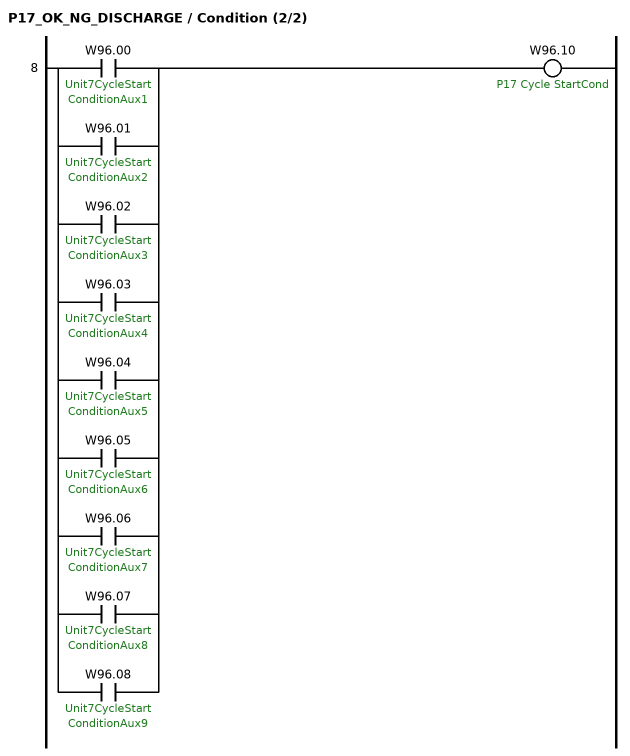
; [picture p288: P17_OK_NG_DISCHARGE / Condition, rungs 8-8]
; rung 8
LD W96.00  ; Unit7CycleStartConditionAux1
OR W96.01  ; Unit7CycleStartConditionAux2
OR W96.02  ; Unit7CycleStartConditionAux3
OR W96.03  ; Unit7CycleStartConditionAux4
OR W96.04  ; Unit7CycleStartConditionAux5
OR W96.05  ; Unit7CycleStartConditionAux6
OR W96.06  ; Unit7CycleStartConditionAux7
OR W96.07  ; Unit7CycleStartConditionAux8
OR W96.08  ; Unit7CycleStartConditionAux9
OUT W96.10  ; P17 Cycle StartCond

### Section Device_Output

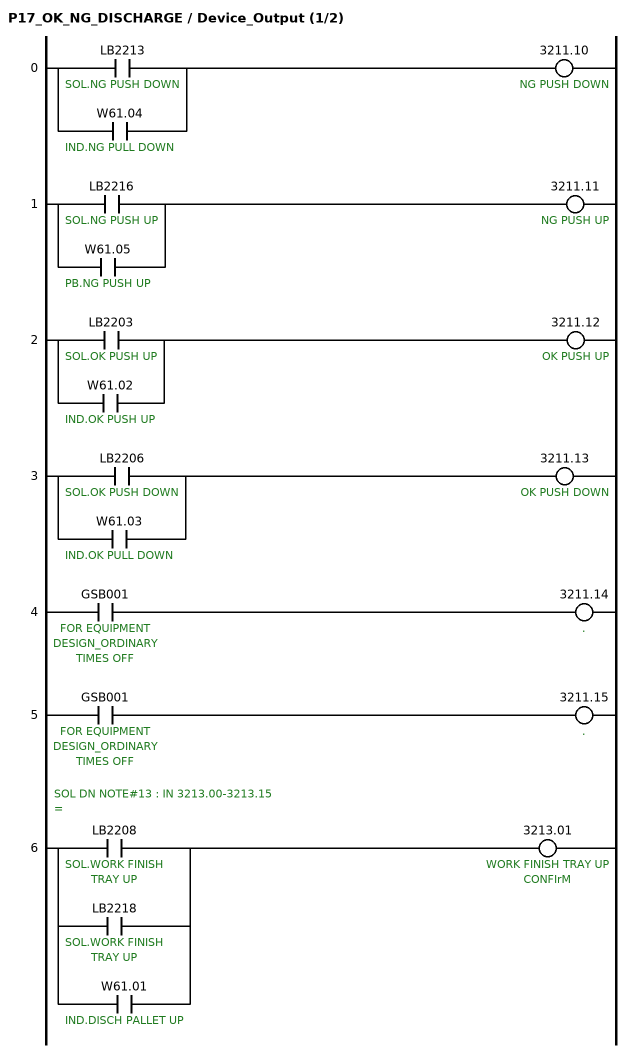
; rung 0
LD LB2213  ; SOL.NG PUSH DOWN
OR W61.04  ; IND.NG PULL DOWN
OUT 3211.10  ; NG PUSH DOWN
; rung 1
LD LB2216  ; SOL.NG PUSH UP
OR W61.05  ; PB.NG PUSH UP
OUT 3211.11  ; NG PUSH UP
; rung 2
LD LB2203  ; SOL.OK PUSH UP
OR W61.02  ; IND.OK PUSH UP
OUT 3211.12  ; OK PUSH UP
; rung 3
LD LB2206  ; SOL.OK PUSH DOWN
OR W61.03  ; IND.OK PULL DOWN
OUT 3211.13  ; OK PUSH DOWN
; rung 4
LD GSB001  ; FOR EQUIPMENT DESIGN_ORDINARY TIMES OFF
OUT 3211.14  ; .
; rung 5
LD GSB001  ; FOR EQUIPMENT DESIGN_ORDINARY TIMES OFF
OUT 3211.15  ; .
; rung 6: SOL DN NOTE#13 : IN 3213.00-3213.15 / =
LD LB2208  ; SOL.WORK FINISH TRAY UP
OR LB2218  ; SOL.WORK FINISH TRAY UP
OR W61.01  ; IND.DISCH PALLET UP
OUT 3213.01  ; WORK FINISH TRAY UP CONFIrM

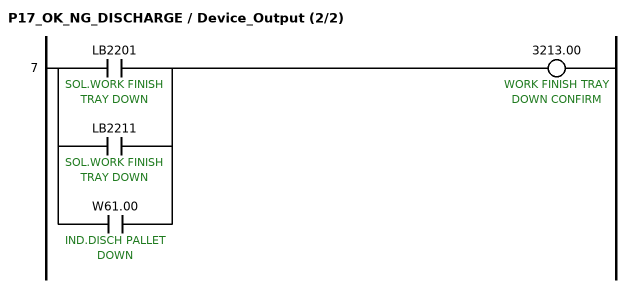
; rung 7
LD LB2201  ; SOL.WORK FINISH TRAY DOWN
OR LB2211  ; SOL.WORK FINISH TRAY DOWN
OR W61.00  ; IND.DISCH PALLET DOWN
OUT 3213.00  ; WORK FINISH TRAY DOWN CONFIRM

### Section Station_Output

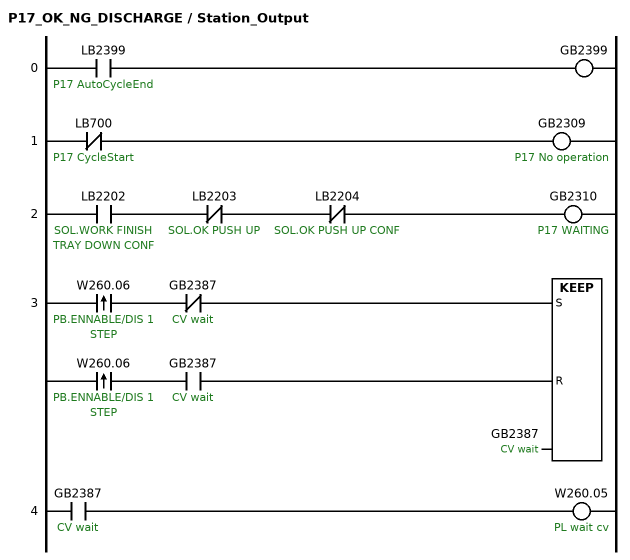
; rung 0
LD LB2399  ; P17 AutoCycleEnd
OUT GB2399
; rung 1
LDNOT LB700  ; P17 CycleStart
OUT GB2309  ; P17 No operation
; rung 2
LD LB2202  ; SOL.WORK FINISH TRAY DOWN CONF
ANDNOT LB2203  ; SOL.OK PUSH UP
ANDNOT LB2204  ; SOL.OK PUSH UP CONF
OUT GB2310  ; P17 WAITING
; rung 3
@LD W260.06  ; PB.ENNABLE/DIS 1 STEP
ANDNOT GB2387  ; CV wait
@LD W260.06  ; PB.ENNABLE/DIS 1 STEP
AND GB2387  ; CV wait
KEEP GB2387  ; CV wait
; rung 4
LD GB2387  ; CV wait
OUT W260.05  ; PL wait cv

### Section Individual

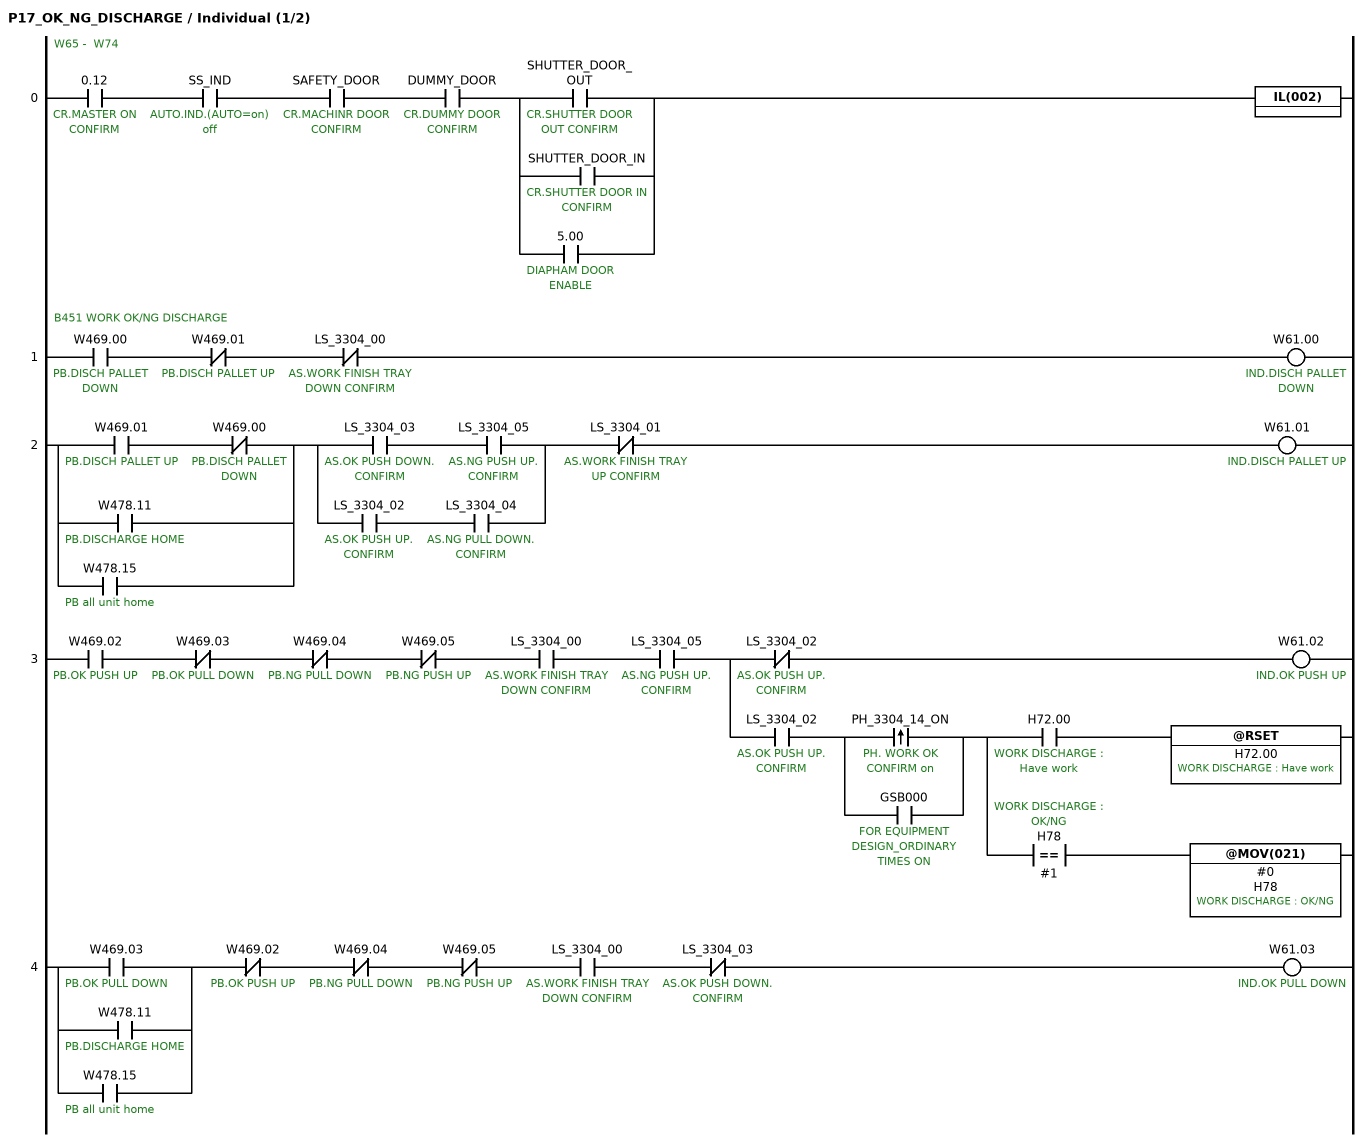
; rung 0: W65 -  W74
LD 0.12  ; CR.MASTER ON CONFIRM
AND SS_IND  ; AUTO.IND.(AUTO=on) off
AND SAFETY_DOOR  ; CR.MACHINR DOOR CONFIRM
AND DUMMY_DOOR  ; CR.DUMMY DOOR CONFIRM
LD SHUTTER_DOOR_OUT  ; CR.SHUTTER DOOR OUT CONFIRM
OR SHUTTER_DOOR_IN  ; CR.SHUTTER DOOR IN CONFIRM
OR 5.00  ; DIAPHAM DOOR ENABLE
ANDLD
IL(002)
; rung 1: B451 WORK OK/NG DISCHARGE
LD W469.00  ; PB.DISCH PALLET DOWN
ANDNOT W469.01  ; PB.DISCH PALLET UP
ANDNOT LS_3304_00  ; AS.WORK FINISH TRAY DOWN CONFIRM
OUT W61.00  ; IND.DISCH PALLET DOWN
; rung 2
LD W469.01  ; PB.DISCH PALLET UP
ANDNOT W469.00  ; PB.DISCH PALLET DOWN
LD W478.11  ; PB.DISCHARGE HOME
OR W478.15  ; PB all unit home
ORLD
LD LS_3304_03  ; AS.OK PUSH DOWN. CONFIRM
AND LS_3304_05  ; AS.NG PUSH UP. CONFIRM
LD LS_3304_02  ; AS.OK PUSH UP. CONFIRM
AND LS_3304_04  ; AS.NG PULL DOWN. CONFIRM
ORLD
ANDLD
ANDNOT LS_3304_01  ; AS.WORK FINISH TRAY UP CONFIRM
OUT W61.01  ; IND.DISCH PALLET UP
; rung 3
LD W469.02  ; PB.OK PUSH UP
ANDNOT W469.03  ; PB.OK PULL DOWN
ANDNOT W469.04  ; PB.NG PULL DOWN
ANDNOT W469.05  ; PB.NG PUSH UP
AND LS_3304_00  ; AS.WORK FINISH TRAY DOWN CONFIRM
AND LS_3304_05  ; AS.NG PUSH UP. CONFIRM
OUT TR0
ANDNOT LS_3304_02  ; AS.OK PUSH UP. CONFIRM
OUT W61.02  ; IND.OK PUSH UP
LD TR0
AND LS_3304_02  ; AS.OK PUSH UP. CONFIRM
@LD PH_3304_14_ON  ; PH. WORK OK CONFIRM on
OR GSB000  ; FOR EQUIPMENT DESIGN_ORDINARY TIMES ON
ANDLD
OUT TR0
AND H72.00  ; WORK DISCHARGE : Have work
@RSET H72.00  ; WORK DISCHARGE : Have work
LD TR0
AND=(300) H78 #1  ; WORK DISCHARGE : OK/NG
@MOV(021) #0 H78  ; WORK DISCHARGE : OK/NG
; rung 4
LD W469.03  ; PB.OK PULL DOWN
OR W478.11  ; PB.DISCHARGE HOME
OR W478.15  ; PB all unit home
ANDNOT W469.02  ; PB.OK PUSH UP
ANDNOT W469.04  ; PB.NG PULL DOWN
ANDNOT W469.05  ; PB.NG PUSH UP
AND LS_3304_00  ; AS.WORK FINISH TRAY DOWN CONFIRM
ANDNOT LS_3304_03  ; AS.OK PUSH DOWN. CONFIRM
OUT W61.03  ; IND.OK PULL DOWN

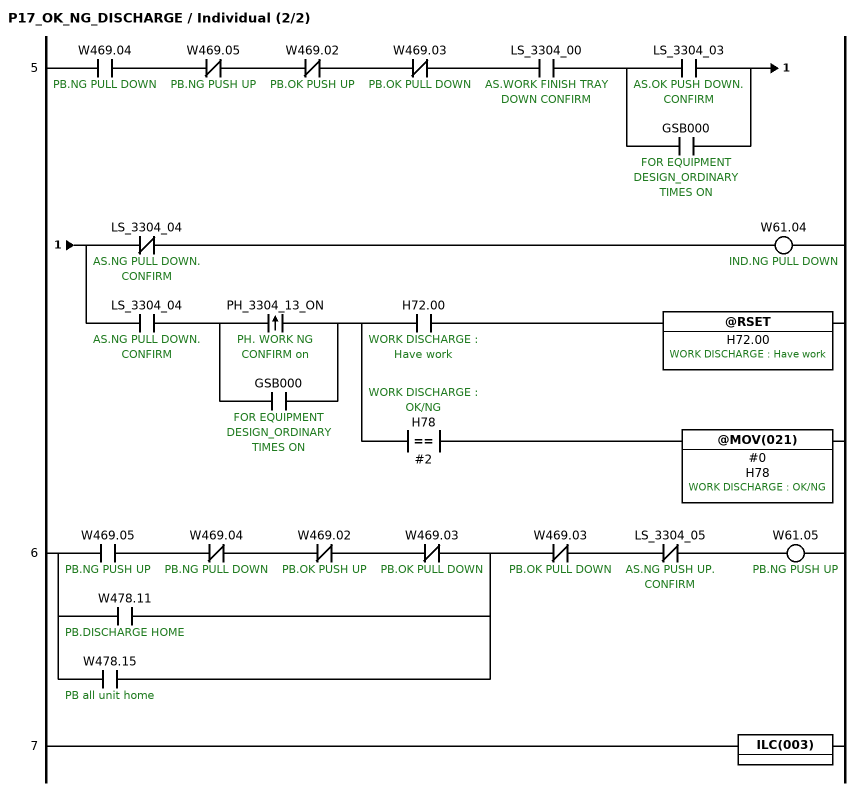
; rung 5
LD W469.04  ; PB.NG PULL DOWN
ANDNOT W469.05  ; PB.NG PUSH UP
ANDNOT W469.02  ; PB.OK PUSH UP
ANDNOT W469.03  ; PB.OK PULL DOWN
AND LS_3304_00  ; AS.WORK FINISH TRAY DOWN CONFIRM
LD LS_3304_03  ; AS.OK PUSH DOWN. CONFIRM
OR GSB000  ; FOR EQUIPMENT DESIGN_ORDINARY TIMES ON
ANDLD
OUT TR0
ANDNOT LS_3304_04  ; AS.NG PULL DOWN. CONFIRM
OUT W61.04  ; IND.NG PULL DOWN
LD TR0
AND LS_3304_04  ; AS.NG PULL DOWN. CONFIRM
@LD PH_3304_13_ON  ; PH. WORK NG CONFIRM on
OR GSB000  ; FOR EQUIPMENT DESIGN_ORDINARY TIMES ON
ANDLD
OUT TR0
AND H72.00  ; WORK DISCHARGE : Have work
@RSET H72.00  ; WORK DISCHARGE : Have work
LD TR0
AND=(300) H78 #2  ; WORK DISCHARGE : OK/NG
@MOV(021) #0 H78  ; WORK DISCHARGE : OK/NG
; rung 6
LD W469.05  ; PB.NG PUSH UP
ANDNOT W469.04  ; PB.NG PULL DOWN
ANDNOT W469.02  ; PB.OK PUSH UP
ANDNOT W469.03  ; PB.OK PULL DOWN
LD W478.11  ; PB.DISCHARGE HOME
OR W478.15  ; PB all unit home
ORLD
ANDNOT W469.03  ; PB.OK PULL DOWN
ANDNOT LS_3304_05  ; AS.NG PUSH UP. CONFIRM
OUT W61.05  ; PB.NG PUSH UP
; rung 7
ILC(003)

### Section HMI_Output

### Section END
; rung 0
END(001)